{attribute 'GeneratedUsingTerminal: IODEVICETYPE_ETHERCATPROT'}
{attribute addProperty BoxType "IODEVICETYPE_ETHERCATPROT"}
{attribute addProperty Id "Beckhoff_EP1xxxBeckhoff_EP1xxx_617026EA1740Beckhoff_EP2xxxBeckhoff_EP2xxx_5E6BC55D3524Beckhoff_EP3xxxBeckhoff_EP3xxx_05483C403196Beckhoff_EP4xxxBeckhoff_EP4xxx_5F57EEFA336Beckhoff_EP5xxxBeckhoff_EP5xxx_7357566B409Beckhoff_EP6xxxBeckhoff_EP6xxx_09B4DFD61410Beckhoff_EP7xxxBeckhoff_EP7xxx_ED3612242992Beckhoff_EP8xxxBeckhoff_EP8xxx_7FC896F3282Beckhoff_EP9xxxBeckhoff_EP9xxx_0E1CA865617SyncUnitsSyncUnits_2E61B95536InputsInputs_25A0042B160OutputsOutputs_2397A10E106InfoDataInfoData_E68C61CD28"}
{attribute addProperty CRC "725847387"}
{attribute addProperty Size "14836"}
TYPE EtherCAT_Master_EPxxxx_2B438D5B :
STRUCT
	{attribute addProperty Name "Beckhoff EP1xxx"}
	{attribute addProperty PreviousPort "EtherCAT_Master_EPxxxx : Master"}
	Beckhoff_EP1xxx : Beckhoff_EP1xxx_617026EA;
	{attribute addProperty Name "Beckhoff EP2xxx"}
	{attribute addProperty PreviousPort "Beckhoff EP1xxx : C"}
	Beckhoff_EP2xxx : Beckhoff_EP2xxx_5E6BC55D;
	{attribute addProperty Name "Beckhoff EP3xxx"}
	{attribute addProperty PreviousPort "Beckhoff EP2xxx : C"}
	Beckhoff_EP3xxx : Beckhoff_EP3xxx_05483C40;
	{attribute addProperty Name "Beckhoff EP4xxx"}
	{attribute addProperty PreviousPort "Beckhoff EP3xxx : C"}
	Beckhoff_EP4xxx : Beckhoff_EP4xxx_5F57EEFA;
	{attribute addProperty Name "Beckhoff EP5xxx"}
	{attribute addProperty PreviousPort "Beckhoff EP4xxx : C"}
	Beckhoff_EP5xxx : Beckhoff_EP5xxx_7357566B;
	{attribute addProperty Name "Beckhoff EP6xxx"}
	{attribute addProperty PreviousPort "Beckhoff EP5xxx : C"}
	Beckhoff_EP6xxx : Beckhoff_EP6xxx_09B4DFD6;
	{attribute addProperty Name "Beckhoff EP7xxx"}
	{attribute addProperty PreviousPort "Beckhoff EP6xxx : C"}
	Beckhoff_EP7xxx : Beckhoff_EP7xxx_ED361224;
	{attribute addProperty Name "Beckhoff EP8xxx"}
	{attribute addProperty PreviousPort "Beckhoff EP7xxx : C"}
	Beckhoff_EP8xxx : Beckhoff_EP8xxx_7FC896F3;
	{attribute addProperty Name "Beckhoff EP9xxx"}
	{attribute addProperty PreviousPort "Beckhoff EP8xxx : C"}
	Beckhoff_EP9xxx : Beckhoff_EP9xxx_0E1CA865;
	{attribute addProperty Name "SyncUnits"}
	SyncUnits : SyncUnits_2E61B955;
	{attribute addProperty Name "Inputs"}
	Inputs : Inputs_25A0042B;
	{attribute addProperty Name "Outputs"}
	Outputs : Outputs_2397A10E;
	{attribute addProperty Name "InfoData"}
	InfoData : InfoData_E68C61CD;
END_STRUCT
END_TYPE

(* stored: Version 1.2.0.0, ProductVersion 3.1.4024.9
   DUT EtherCAT_Master_EPxxxx_2B438D5B: Id {d00172ce-f54c-4481-b4e3-7760e3f3b61b} *)
